(* PLC project switch_3pos_2outputs, Dassault Systèmes ControlBuild 2024x *)
(* stored: creationDateTime 2023-10-03T11:13:22-01:00 *)

(* This module simulates a switch with 3 positions and 2 outputs. *)
FUNCTION_BLOCK equipment_library.switch_3pos_2outputs
  VAR_OUTPUT
    leftVariable : BOOL := false;
    rightVariable : BOOL := false;
  END_VAR
  VAR
    leftPosition : BOOL := false;
    middlePosition : BOOL := false;
    rightPosition : BOOL := false;
  END_VAR

(* -----------------------------------------------------------------	*)
(* Type : Model of Operative Behaviour					*)
(* Category :  Power								*)
(* Author : Dassault Systemes						*)
(* Update date : June 2018							*)
(* -----------------------------------------------------------------	*)
(* This module simulates a switch with 3 positions and 2 outputs.	*)
(* -----------------------------------------------------------------	*)

IF (leftPosition) THEN
	leftVariable := TRUE;
	rightVariable := FALSE;
END_IF;
IF (middlePosition) THEN
	leftVariable := FALSE;
	rightVariable := FALSE;
END_IF;
IF (rightPosition) THEN
	leftVariable := FALSE;
	rightVariable := TRUE;
END_IF;
leftPosition := FALSE;
middlePosition := FALSE;
rightPosition := FALSE;
END_FUNCTION_BLOCK
